INTERFACE I_InputPorts

METHOD PUBLIC GetEnumerator : I_ForwardEnumerator
VAR_INPUT
END_VAR
END_METHOD

METHOD PUBLIC TryGetByName : BOOL;
VAR_INPUT
	Name : STRING;
	Destination : REFERENCE TO I_InputPort;
END_VAR
END_METHOD

END_INTERFACE

(* stored: Version 1.1.0.1, ProductVersion 3.1.4024.12
   Itf I_InputPorts: Id {94227c78-86cf-000d-3859-5ce8c7e6b5ed}
   Method GetEnumerator: Id {90c5fafc-11b0-0611-02f9-b83a25964a95}
   Method TryGetByName: Id {e27f268e-ec73-0dfb-0dee-7995d92aefeb} *)
